(* IEC 61131-3 sources: repolevel_ST_code_completion/dataset/project_code/Command1/FUN, 38 files *)

(* ---- FB_AirConComfortCommand.st ---- *)
FUNCTION_BLOCK PUBLIC FB_AirConComfortCommand IMPLEMENTS I_Command
VAR
	refAirConditioning : REFERENCE TO FB_AirConditioning;
END_VAR

(* ---- FB_AirConditioning.st ---- *)
FUNCTION_BLOCK PUBLIC FB_AirConditioning
VAR_OUTPUT
	bActive			: BOOL;
	lrTemperature	: LREAL;
END_VAR

(* ---- FB_AirConStandbyCommand.st ---- *)
FUNCTION_BLOCK PUBLIC FB_AirConStandbyCommand IMPLEMENTS I_Command
VAR
	refAirConditioning : REFERENCE TO FB_AirConditioning;
END_VAR

(* ---- FB_CDPlayer.st ---- *)
FUNCTION_BLOCK PUBLIC FB_CDPlayer
VAR_OUTPUT
	bPlayerActive		: BOOL;
	byVolume			: BYTE;
	byTrack				: UINT;
END_VAR

(* ---- FB_Lamp.st ---- *)
FUNCTION_BLOCK PUBLIC FB_Lamp
VAR_OUTPUT
	byLevel			: BYTE;
END_VAR

(* ---- FB_LampSetLevelCommand.st ---- *)
FUNCTION_BLOCK PUBLIC FB_LampSetLevelCommand IMPLEMENTS I_Command
VAR
	refLamp		: REFERENCE TO FB_Lamp;
	byNewLevel	: BYTE;
END_VAR

(* ---- FB_MusicPlayCommand.st ---- *)
FUNCTION_BLOCK PUBLIC FB_MusicPlayCommand IMPLEMENTS I_Command
VAR
	refCDPlayer : REFERENCE TO FB_CDPlayer;
END_VAR

(* ---- FB_MusicStopCommand.st ---- *)
FUNCTION_BLOCK PUBLIC FB_MusicStopCommand IMPLEMENTS I_Command
VAR
	refCDPlayer : REFERENCE TO FB_CDPlayer;
END_VAR

(* ---- FB_Socket.st ---- *)
FUNCTION_BLOCK PUBLIC FB_Socket
VAR_OUTPUT
	bActive		: BOOL;
END_VAR

(* ---- FB_SocketOffCommand.st ---- *)
FUNCTION_BLOCK PUBLIC FB_SocketOffCommand IMPLEMENTS I_Command
VAR
	refSocket : REFERENCE TO FB_Socket;
END_VAR

(* ---- FB_SocketOffCommand_FB_init.st ---- *)
FUNCTION_BLOCK PUBLIC FB_AirConStandbyCommand IMPLEMENTS I_Command
VAR
	refSocket : REFERENCE TO FB_Socket;
END_VAR
VAR_INPUT
	bInitRetains : BOOL; // if TRUE, the retain variables are initialized (warm start / cold start)
	bInCopyCode : BOOL;  // if TRUE, the instance afterwards gets moved into the copy code (online change)
	refNewSocket : REFERENCE TO FB_Socket;
END_VAR

IF (__ISVALIDREF(refNewSocket)) THEN
	THIS^.refSocket REF= refNewSocket;
ELSE
	THIS^.refSocket REF= 0;
END_IF

(* ---- FB_SocketOnCommand.st ---- *)
FUNCTION_BLOCK PUBLIC FB_SocketOnCommand IMPLEMENTS I_Command
VAR
	refSocket : REFERENCE TO FB_Socket;
END_VAR

(* ---- FB_SwitchPanel.st ---- *)
FUNCTION_BLOCK PUBLIC FB_SwitchPanel
VAR_INPUT
	arrSwitch		: ARRAY[1..8] OF BOOL;
END_VAR
VAR
	aiCommand		: ARRAY[1..8] OF I_Command;
	arrRtrig		: ARRAY[1..8] OF R_TRIG;
	nIndex			: INT;
END_VAR

FOR nIndex := 1 TO 8 DO
	arrRtrig[nIndex](CLK := arrSwitch[nIndex]);
	IF arrRtrig[nIndex].Q THEN
		IF (aiCommand[nIndex] <> 0) THEN
			aiCommand[nIndex].Execute();
		END_IF
	END_IF
END_FOR

(* ---- FB_AirConComfortCommand_Execute.st ---- *)
METHOD Execute
VAR
	refAirConditioning : REFERENCE TO FB_AirConditioning;
END_VAR

IF (__ISVALIDREF(THIS^.refAirConditioning)) THEN
	THIS^.refAirConditioning.Activate();
	THIS^.refAirConditioning.SetTemperature(20.0);
END_IF

(* ---- FB_AirConComfortCommand_FB_init.st ---- *)
METHOD FB_init : BOOL
VAR_INPUT
	bInitRetains : BOOL; // if TRUE, the retain variables are initialized (warm start / cold start)
	bInCopyCode : BOOL;  // if TRUE, the instance afterwards gets moved into the copy code (online change)
	refAirConditioning : REFERENCE TO FB_AirConditioning;
END_VAR
VAR
	refAirConditioning : REFERENCE TO FB_AirConditioning;
END_VAR

IF (__ISVALIDREF(refAirConditioning)) THEN
	THIS^.refAirConditioning REF= refAirConditioning;
ELSE
	THIS^.refAirConditioning REF= 0;
END_IF

(* ---- FB_AirConditioning_Activate.st ---- *)
METHOD PUBLIC Activate
VAR_OUTPUT
	bActive			: BOOL;
	lrTemperature	: LREAL;
END_VAR

bActive := TRUE;

(* ---- FB_AirConditioning_Deactivate.st ---- *)
METHOD PUBLIC Deactivate
VAR_OUTPUT
	bActive			: BOOL;
	lrTemperature	: LREAL;
END_VAR

bActive := false;

(* ---- FB_AirConditioning_SetTemperature.st ---- *)
METHOD PUBLIC SetTemperature : BOOL
VAR_INPUT
	lrNewTemperature	: LREAL;
END_VAR
VAR_OUTPUT
	bActive			: BOOL;
	lrTemperature	: LREAL;
END_VAR

lrTemperature := lrNewTemperature;

(* ---- FB_AirConStandbyCommand_Execute.st ---- *)
METHOD Execute
VAR
	refAirConditioning : REFERENCE TO FB_AirConditioning;
END_VAR

IF (__ISVALIDREF(THIS^.refAirConditioning)) THEN
	THIS^.refAirConditioning.Activate();
	THIS^.refAirConditioning.SetTemperature(17.5);
END_IF

(* ---- FB_AirConStandbyCommand_FB_init.st ---- *)
METHOD FB_init : BOOL
VAR_INPUT
	bInitRetains : BOOL; // if TRUE, the retain variables are initialized (warm start / cold start)
	bInCopyCode : BOOL;  // if TRUE, the instance afterwards gets moved into the copy code (online change)
	refAirConditioning : REFERENCE TO FB_AirConditioning;
END_VAR
VAR
	refAirConditioning : REFERENCE TO FB_AirConditioning;
END_VAR

IF (__ISVALIDREF(refAirConditioning)) THEN
	THIS^.refAirConditioning REF= refAirConditioning;
ELSE
	THIS^.refAirConditioning REF= 0;
END_IF

(* ---- FB_CDPlayer_setTrack.st ---- *)
METHOD PUBLIC SetTrack : BOOL
VAR_INPUT
	byNewTrack			: UINT;
END_VAR
VAR_OUTPUT
	bPlayerActive		: BOOL;
	byVolume			: BYTE;
	byTrack				: UINT;
END_VAR

byTrack := byNewTrack;

(* ---- FB_CDPlayer_setVolume.st ---- *)
METHOD PUBLIC SetVolume : BOOL
VAR_INPUT
	byNewVolume 		: BYTE;
END_VAR
VAR_OUTPUT
	bPlayerActive		: BOOL;
	byVolume			: BYTE;
	byTrack				: UINT;
END_VAR

byVolume := byNewVolume;

(* ---- FB_CDPlayer_Start.st ---- *)
METHOD PUBLIC Start
VAR_OUTPUT
	bPlayerActive		: BOOL;
	byVolume			: BYTE;
	byTrack				: UINT;
END_VAR

bPlayerActive := true;

(* ---- FB_CDPlayer_Stop.st ---- *)
METHOD PUBLIC Stop
VAR_OUTPUT
	bPlayerActive		: BOOL;
	byVolume			: BYTE;
	byTrack				: UINT;
END_VAR

bPlayerActive := FALSE;

(* ---- FB_Lamp_SetLevel.st ---- *)
METHOD PUBLIC SetLevel : BOOL
VAR_OUTPUT
	byLevel			: BYTE;
END_VAR
VAR_INPUT
	byNewLevel			: BYTE;
END_VAR
byLevel := byNewLevel;

(* ---- FB_LampSetLevelCommand_Execute.st ---- *)
METHOD Execute
VAR
	refAirConditioning : REFERENCE TO FB_AirConditioning;
END_VAR

IF (__ISVALIDREF(THIS^.refLamp)) THEN
	THIS^.refLamp.SetLevel(THIS^.byNewLevel);
END_IF

(* ---- FB_LampSetLevelCommand_FB_init.st ---- *)
METHOD FB_init : BOOL
VAR_INPUT
	bInitRetains : BOOL; // if TRUE, the retain variables are initialized (warm start / cold start)
	bInCopyCode : BOOL;  // if TRUE, the instance afterwards gets moved into the copy code (online change)
	refLamp : REFERENCE TO FB_Lamp;
	byNewLevel : BYTE;
END_VAR
VAR
	refLamp		: REFERENCE TO FB_Lamp;
	byNewLevel	: BYTE;
END_VAR

IF (__ISVALIDREF(refLamp)) THEN
	THIS^.refLamp REF= refLamp;
ELSE
	THIS^.refLamp REF= 0;
END_IF
THIS^.byNewLevel := byNewLevel;

(* ---- FB_MusicPlayCommand_Execute.st ---- *)
METHOD Execute
VAR
	refCDPlayer : REFERENCE TO FB_CDPlayer;
END_VAR

IF (__ISVALIDREF(THIS^.refCDPlayer)) THEN
	THIS^.refCDPlayer.SetVolume(40);
	THIS^.refCDPlayer.SetTrack(1);
	THIS^.refCDPlayer.Start();
END_IF

(* ---- FB_MusicPlayCommand_FB_init.st ---- *)
METHOD FB_init : BOOL
VAR_INPUT
	bInitRetains : BOOL; // if TRUE, the retain variables are initialized (warm start / cold start)
	bInCopyCode : BOOL;  // if TRUE, the instance afterwards gets moved into the copy code (online change)
	refCDPlayer : REFERENCE TO FB_CDPlayer;
END_VAR
VAR
	refCDPlayer : REFERENCE TO FB_CDPlayer;
END_VAR

IF (__ISVALIDREF(refCDPlayer)) THEN
	THIS^.refCDPlayer REF= refCDPlayer;
ELSE
	THIS^.refCDPlayer REF= 0;
END_IF

(* ---- FB_MusicStopCommand_Execute.st ---- *)
METHOD Execute
VAR
	refCDPlayer : REFERENCE TO FB_CDPlayer;
END_VAR

IF (__ISVALIDREF(THIS^.refCDPlayer)) THEN
	THIS^.refCDPlayer.Stop();
END_IF

(* ---- FB_MusicStopCommand_FB_init.st ---- *)
METHOD FB_init : BOOL
VAR_INPUT
	bInitRetains : BOOL; // if TRUE, the retain variables are initialized (warm start / cold start)
	bInCopyCode : BOOL;  // if TRUE, the instance afterwards gets moved into the copy code (online change)
	refCDPlayer : REFERENCE TO FB_CDPlayer;
END_VAR
VAR
	refCDPlayer : REFERENCE TO FB_CDPlayer;
END_VAR

IF (__ISVALIDREF(refCDPlayer)) THEN
	THIS^.refCDPlayer REF= refCDPlayer;
ELSE
	THIS^.refCDPlayer REF= 0;
END_IF

(* ---- FB_Socket_Off.st ---- *)
METHOD PUBLIC Off
VAR_OUTPUT
	bActive		: BOOL;
END_VAR

bActive := false;

(* ---- FB_Socket_On.st ---- *)
METHOD PUBLIC On
VAR_OUTPUT
	bActive		: BOOL;
END_VAR

bActive := true;

(* ---- FB_SocketOffCommand_Execute.st ---- *)
METHOD Execute
VAR
	refSocket : REFERENCE TO FB_Socket;
END_VAR
IF (__ISVALIDREF(THIS^.refSocket)) THEN
	THIS^.refSocket.On();
END_IF

(* ---- FB_SocketOnCommand_Execute.st ---- *)
METHOD Execute
VAR
	refSocket : REFERENCE TO FB_Socket;
END_VAR
IF (__ISVALIDREF(THIS^.refSocket)) THEN
	THIS^.refSocket.On();
END_IF

(* ---- FB_SocketOnCommand_FB_init.st ---- *)
METHOD FB_init : BOOL
VAR_INPUT
	bInitRetains : BOOL; // if TRUE, the retain variables are initialized (warm start / cold start)
	bInCopyCode : BOOL;  // if TRUE, the instance afterwards gets moved into the copy code (online change)
	refNewSocket : REFERENCE TO FB_Socket;
END_VAR
VAR
	refSocket : REFERENCE TO FB_Socket;
END_VAR

IF (__ISVALIDREF(refNewSocket)) THEN
	THIS^.refSocket REF= refNewSocket;
ELSE
	THIS^.refSocket REF= 0;
END_IF

(* ---- FB_SwitchPanel_FB_init.st ---- *)
METHOD FB_init : BOOL
VAR_INPUT
	bInitRetains : BOOL; // if TRUE, the retain variables are initialized (warm start / cold start)
	bInCopyCode : BOOL;  // if TRUE, the instance afterwards gets moved into the copy code (online change)
    arrSwitch		: ARRAY[1..8] OF BOOL;
END_VAR
VAR
	nIndex : INT;
    aiCommand		: ARRAY[1..8] OF I_Command;
	arrRtrig		: ARRAY[1..8] OF R_TRIG;
	nIndex			: INT;
END_VAR

FOR nIndex := 1 TO 8 DO
	aiCommand[nIndex] := 0;
END_FOR

(* ---- FB_SwitchPanel_SetCommand.st ---- *)
METHOD PUBLIC SetCommand : BOOL
VAR_INPUT
	nPosition		: INT;
	iCommand		: I_Command;
    arrSwitch		: ARRAY[1..8] OF BOOL;

END_VAR
VAR
	aiCommand		: ARRAY[1..8] OF I_Command;
	arrRtrig		: ARRAY[1..8] OF R_TRIG;
	nIndex			: INT;
END_VAR

IF ((nPosition >= 1) AND (nPosition <= 8) AND (iCommand <> 0)) THEN
	THIS^.aiCommand[nPosition] := iCommand;
END_IF
